// LS Electric XG5000 project: 7-모터수증감
// PLC NewPLC
// module base 0 slot 0: 입출력 모듈:XBC-DN/DP14E (DC 24V 입력 8점, 트랜지스터 출력 6점)

PROGRAM NewProgram (task: 스캔 프로그램)

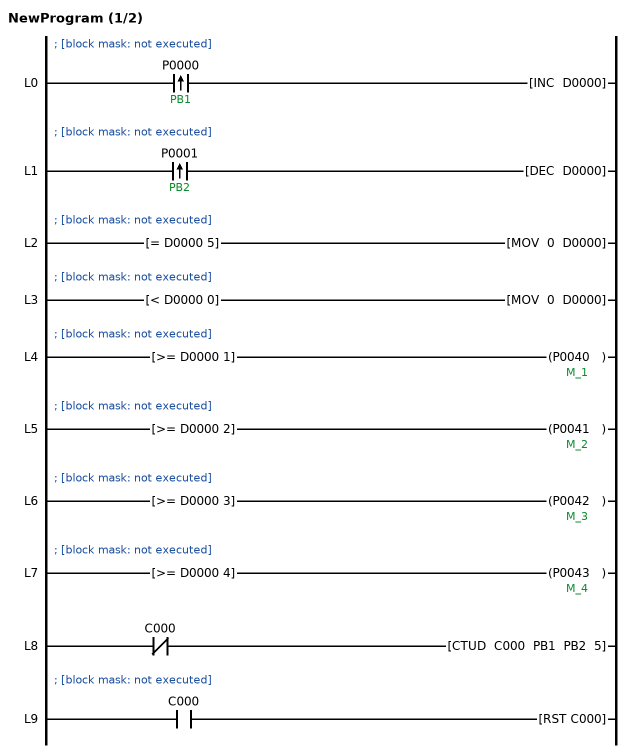
; L0 (block mask: not executed)
LOADP     P0000	// PB1
INC       D0000
; L1 (block mask: not executed)
LOADP     P0001	// PB2
DEC       D0000
; L2 (block mask: not executed)
LOAD=     D0000 5
MOV       0 D0000
; L3 (block mask: not executed)
LOAD<     D0000 0
MOV       0 D0000
; L4 (block mask: not executed)
LOAD>=    D0000 1
OUT       P0040	// M_1
; L5 (block mask: not executed)
LOAD>=    D0000 2
OUT       P0041	// M_2
; L6 (block mask: not executed)
LOAD>=    D0000 3
OUT       P0042	// M_3
; L7 (block mask: not executed)
LOAD>=    D0000 4
OUT       P0043	// M_4
; L8
LOAD NOT  C000
CTUD      C000 PB1 PB2 5
; L9 (block mask: not executed)
LOAD      C000
RST       C000

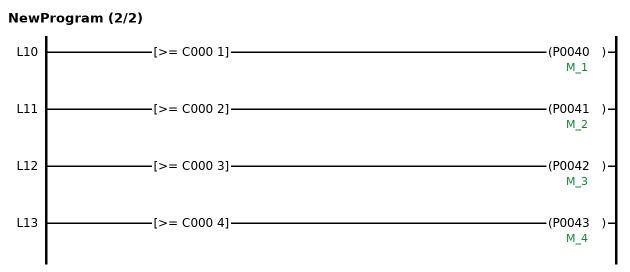
; L10
LOAD>=    C000 1
OUT       P0040	// M_1
; L11
LOAD>=    C000 2
OUT       P0041	// M_2
; L12
LOAD>=    C000 3
OUT       P0042	// M_3
; L13
LOAD>=    C000 4
OUT       P0043	// M_4